TYPE ST_Syntax_ExhaustiveArrays :
STRUCT
    arrStaticInts   : ARRAY[1..8] OF INT := [1, 2, 3, 4, 5, 6, 7, 8];
    arrMultiDimInt  : ARRAY[1..2, 1..2] OF INT;
    arrMultilineInt : ARRAY[1..4] OF INT := [
        1, 2,
        3, 4
    ];
    arrNestedMini   : ARRAY[1..2] OF ST_Syntax_Mini := [
        (nId := 1, bActive := TRUE, sName := 'SubA'),
        (nId := 2, bActive := FALSE, sName := 'SubB')
    ];
END_STRUCT
END_TYPE

(* stored: Version 1.1.0.1, ProductVersion 3.1.4024.16
   DUT ST_Syntax_ExhaustiveArrays: Id {b6e9035c-4d2f-4610-8340-f90d7340cd82} *)
